{attribute 'qualified_only'}
VAR_GLOBAL
	waferInspectionRecipe : WaferInspection;
	Camera : SimpleCamera;
	LabelProcess : ProcessSKU;
	ImageChannel : VisionChannel(Name := 'Beckhoff Camera', ImageSource := Camera, ImageProcess := LabelProcess);
END_VAR

(* stored: Version 1.1.0.1
   GVL GVL_Vision: Id {fb719938-f404-4796-9ddd-b170432ceb2f} *)
